{attribute 'hide_all_locals'}
FUNCTION_BLOCK PUBLIC ABSTRACT FB_Employee
VAR_INPUT
END_VAR
VAR_OUTPUT
END_VAR
VAR
	nPersonnelNumberBacking :	UINT;
	sFirstNameBacking		:	STRING;
	sLastNameBacking		:	STRING;
END_VAR

METHOD PUBLIC GetFullName : STRING
VAR_INPUT
END_VAR
GetFullName := CONCAT(CONCAT(CONCAT(CONCAT(TO_STRING(nPersonnelNumber), ': '), sFirstName), ' '), sLastName);
END_METHOD

METHOD PUBLIC ABSTRACT GetMonthlySalary : LREAL
VAR_INPUT
END_VAR
END_METHOD

{attribute 'monitoring' := 'variable'}
PROPERTY PUBLIC nPersonnelNumber : UINT
GET
nPersonnelNumber := nPersonnelNumberBacking;
END_GET
SET
nPersonnelNumberBacking := nPersonnelNumber;
END_SET
END_PROPERTY

{attribute 'monitoring' := 'variable'}
PROPERTY PUBLIC sFirstName : STRING
GET
sFirstName := sFirstNameBacking;
END_GET
SET
sFirstNameBacking := sFirstName;
END_SET
END_PROPERTY

{attribute 'monitoring' := 'variable'}
PROPERTY PUBLIC sLastName : STRING
GET
sLastName := sLastNameBacking;
END_GET
SET
sLastNameBacking := sLastName;
END_SET
END_PROPERTY

END_FUNCTION_BLOCK

(* stored: Version 1.1.0.1, ProductVersion 3.1.4024.4
   POU FB_Employee: Id {2cc7defd-3e09-4270-815e-92d7c2b9e2ed}, SpecialFunc None
   Method GetFullName: Id {a38adcfd-bdb3-4984-8ca9-9695a28e2a21}
   Method GetMonthlySalary: Id {c2c84659-4bba-4b37-8367-127abc5f70e0}
   Property nPersonnelNumber: Id {7eca07d9-ded1-4ef4-8f6f-f1a39ae6d112}
   Get Get: Id {45cb952b-d08c-432a-9b00-a30c0f77f415}
   Set Set: Id {1461992f-b159-410f-a337-588f492a8ad2}
   Property sFirstName: Id {b4a086ca-225d-476d-8efa-e89be1aaab40}
   Get Get: Id {3c6d8eff-8379-4af7-8d88-01855bd1750b}
   Set Set: Id {142ffc25-5e82-4e0a-924f-4113b6068e07}
   Property sLastName: Id {2b72463c-3390-4d6c-b808-2f94b0f06cc4}
   Get Get: Id {73ca322d-46f6-4d3a-bed9-a6472e6f71e5}
   Set Set: Id {0e0a4780-ed7c-48ca-9d8b-94c8b1e5b22e} *)
